TYPE ST_ModbusDeviceParam :
STRUCT
	MBSAdress			: BYTE	:= 30;
	UpdateTime			: TIME	:= T#1000MS;
END_STRUCT
END_TYPE

(* stored: Version 1.1.0.1
   DUT ST_ModbusDeviceParam: Id {eea7bccf-a1f2-4c59-b0fd-5dd76c92d4b9} *)
